PROGRAM P_VCB
VAR
	eSwitch : E_Mode;
	fbModeSelect : FB_ModeSelect;
	fbStatus : FB_Status;
END_VAR

fbModeSelect();

fbStatus(
bFault := HMI.stVisuParam.bFault,
bStart:= HMI.stVisuParam.bStart,
bStop := HMI.stVisuParam.bStop,
bRunning := HMI.stVisuParam.bRunning,
eStatus => HMI.eStatus,
bAuto := HMI.stVisuParam.bAuto,
bOn := HMI.stVisuParam.bOn
);

END_PROGRAM

(* stored: Version 1.1.0.1, ProductVersion 3.1.4024.12
   POU P_VCB: Id {ded2fcc5-1dd9-4ee2-b935-1315ce93d88c}, SpecialFunc None *)
